PROGRAM MAIN
VAR
END_VAR


EVACUAZIONE_SCARTI();


//RULLI_CENTRO_TAGLI();

//GESTIONE_ASSI();

END_PROGRAM

(* stored: Version 1.1.0.1, ProductVersion 3.1.4022.12
   POU MAIN: Id {ca1c6c62-0a48-4011-896f-be9b8f84745f}, SpecialFunc None *)
